// TwinCAT 3 PLC project Trappenhuis_Extraverlenging
// ProgramVersion: 3.1.4024.0
// libraries:
//   Tc2_Standard, * (Beckhoff Automation GmbH)
//   Tc2_System, * (Beckhoff Automation GmbH)
//   Tc3_Module, * (Beckhoff Automation GmbH)
// project tree:
//   / PlcTask.TcTTO
//   POUs/ MAIN.TcPOU
// real-time tasks:
//   TASK PlcTask: cycle T#10ms, priority 20, ADS port 350
//   TASK PlcTask1: cycle T#10ms, priority 21, ADS port 351
//   TASK PlcTask2: cycle T#10ms, priority 22, ADS port 352
//   TASK PlcTask3: cycle T#10ms, priority 23, ADS port 353
//   TASK PlcTask4: cycle T#10ms, priority 24, ADS port 354
//   TASK PlcTask5: cycle T#10ms, priority 25, ADS port 355
//   TASK PlcTask6: cycle T#10ms, priority 26, ADS port 356
//   TASK PlcTask7: cycle T#10ms, priority 27, ADS port 357
//   TASK PlcTask8: cycle T#10ms, priority 28, ADS port 358
//   TASK PlcTask9: cycle T#10ms, priority 29, ADS port 359
//   TASK PlcTask10: cycle T#10ms, priority 30, ADS port 360

CONFIGURATION Trappenhuis_Extraverlenging
    RESOURCE PLC ON TwinCAT3
        TASK PlcTask(INTERVAL := T#10ms, PRIORITY := 20);
        PROGRAM MAIN WITH PlcTask : MAIN;
    END_RESOURCE
END_CONFIGURATION

// ---- POUs/MAIN.TcPOU
PROGRAM MAIN
VAR
	// Ingangen
	bDK1               AT %I*: BOOL;
	bDK2               AT %I*: BOOL;
	bDK3               AT %I*: BOOL;
	bDK4               AT %I*: BOOL;
	bDK5               AT %I*: BOOL;
	bDK6               AT %I*: BOOL;
	
	// Uitgangen 
	lamp				AT %Q*: BOOL;
	
	// Timer
	Timer1: TOF;
END_VAR

(*
Trappenhuisautomaat met extra verlenging (1 regel)

In een appartementsgebouw staan in de traphal op de verschillende verdiepingen in totaal 6 drukknoppen. 
Als men één van de drukknoppen bedient gaat de verlichting branden. 
De verlichting blijft 3min. branden - tijdens de test gebruikt men 3s - vooraleer deze vanzelf uitschakelt.
Bij iedere bediening van een drukknop zal de tijd terug beginnen te lopen vanaf 0 en blijven de lampen branden tot de ingestelde tijd is afgelopen.
*)

Timer1(IN:=bDK1 OR bDK2 OR bDK3 OR bDK4 OR bDK5 OR bDK6 ,PT:=T#3s , Q=> lamp, ET=> );

END_PROGRAM
